Staubli VAL3: F4_DELT.pgx

program F4_DELT()
begin
  //delay(10)
  delay(0.5)
  while size(sString)>1
    $ddel(sString,size(sString)-1)
  endWhile
  while size(nPulse)>1
    $ddel(nPulse,size(nPulse)-1)
  endWhile
  while size(pfrmCad)>1
    $ddel(pfrmCad,size(pfrmCad)-1)
  endWhile
  //sScrPts="NOT READY**"
  //bTxtPrSv=false
  bTxtPrSv=false
  sScrPts="NOT READY**"
  //n_sTxt=0
  n_sTxt=0
  call hmi_refreshmain()
end
